FUNCTION_BLOCK FB_Bloque
VAR_INPUT
	Tcheck: TIME := T#1S;
	Treset: TIME := T#1S;
	Tdesplazador: TIME := T#1S;
	Tcinta: TIME := T#0.5S;
END_VAR
VAR_OUTPUT
END_VAR
VAR
	Ciclos: INT;
	Aceptados:INT;
	Rechazados: INT;
	Restantes: INT;
	
	pieza_ok: BOOL;
	
	//Terminal 2
	Pulsador_parada_emergencia AT %I*: BOOL;
	Selector_modo_manual AT %I*: BOOL;
	Pulsador_marcha AT %I*: BOOL;
	Pulsador_parada_NC AT %I*: BOOL;
	Parte_operativa_conectada AT %I*: BOOL;
	Presencia_pale AT %I*: BOOL;
	Codigo_pale_bit_0 AT %I*: BOOL;
	Codigo_pale_bit_1 AT %I*: BOOL;
	
	
	//Terminal 3
	Codigo_pale_bit_2 AT %I*: BOOL;
	Detector_presion AT %I*: BOOL;
	
	//Terminal 4
	Desconecta_parte_operativa AT %Q*: BOOL;
	Lampara_alarma AT %Q*: BOOL;
	Lampara_marcha AT %Q*: BOOL;
	Lampara_falta_material AT %Q*: BOOL;
	Activa_marcha_motor_cinta AT %Q*: BOOL;
	Invierte_marcha_motor_cinta AT %Q*: BOOL;
	Retenedor_pale_baja AT %Q*: BOOL;
	Separador_pale_sube AT %Q*: BOOL;
	
	
	//Terminal 5
 	Avisador_sonoro AT %Q*: BOOL;
	
	//Terminal 6
	Horizontal_descargador_detras AT %I*: BOOL;
	Horizontal_descargador_delante AT %I*: BOOL;
	Vertical_descargador_arriba AT %I*: BOOL;
	Vertical_descargador_abajo AT %I*: BOOL;
	Verificador_arriba AT %I*: BOOL;
	Verificador_abajo AT %I*: BOOL;
	Desplazador_detras AT %I*: BOOL;
	Alimentador_detras AT %I*: BOOL;
	
	
	//Terminal 7
	Alimentador_delante AT %I*: BOOL;
	Vacio_obtenido_vacuostato_descargador AT %I*: BOOL;
	Base_en_Alimentador AT %I*: BOOL;
	
	//Terminal 8
	Descargador_adelante AT %Q*: BOOL;
	Descargador_atras AT %Q*: BOOL;
	Descargador_baja AT %Q*: BOOL;
	Rechazador_adelante AT %Q*: BOOL;
	Verificador_baja AT %Q*: BOOL;
	Desplazador_adelante AT %Q*: BOOL;
	Alimentador_adelante AT %Q*: BOOL;
	Eyector_succiona AT %Q*: BOOL;
	
END_VAR

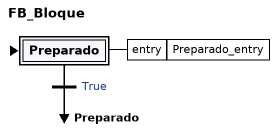
INITIAL_STEP Preparado:
    Preparado_entry(P1);  // entry action
END_STEP
TRANSITION FROM Preparado TO Preparado
    := True;
END_TRANSITION

ACTION notOK_exit:
pieza_ok := FALSE;
END_ACTION

ACTION OK_exit:
pieza_ok := true;
END_ACTION

ACTION Preparado_entry:
//Ciclos:= 3;
Rechazados :=0;
Aceptados :=0;
Restantes:=Ciclos;
END_ACTION

ACTION Rechaza_exit:
Rechazados:= Rechazados+1;
END_ACTION

ACTION Step1_exit:
Ciclos:=Ciclos-1;
Aceptados:=Aceptados+1;
Restantes:=Restantes-1;
END_ACTION

END_FUNCTION_BLOCK

(* stored: Version 1.1.0.1, ProductVersion 3.1.4024.12
   POU FB_Bloque: Id {0c102bf0-d2ee-4790-8611-bbcb80572984}, SpecialFunc None
   Action notOK_exit: Id {7c7983fe-474f-4382-8939-3f4e8ea06912}
   Action OK_exit: Id {6923b980-9502-4e1c-97e4-e82bb8b6c6b3}
   Action Preparado_entry: Id {304360c9-4dcf-4b7e-9bf1-3317d2c36270}
   Action Rechaza_exit: Id {8ccff171-5b8c-4f3f-b00b-570fce4abd22}
   Action Step1_exit: Id {4c99de15-c4a8-4ce6-a026-b728c1b7c456} *)
